(* IEC 61131-3 sources: myrep/src, 2 files *)

(* ---- configuration.st ---- *)
CONFIGURATION MyConfiguration
    TASK Main(Interval := T#1000ms, Priority := 1);
    PROGRAM P1 WITH Main: MyProgram;

    VAR_GLOBAL
        In AT %IW0 : INT;
        Out AT %QW2 : INT;
    END_VAR
END_CONFIGURATION

(* ---- program.st ---- *)
PROGRAM MyProgram
    VAR_EXTERNAL
        In : INT;
        Out : INT;
    END_VAR

    VAR

    END_VAR

    VAR_TEMP

    END_VAR

    // code here
    Out := In;
END_PROGRAM
